TYPE MNG_RawDatagram :
STRUCT
	/// datagram header 
	Header: MNG_DatagramHeader;
	Payload: MNG_DataARRAY;
END_STRUCT
END_TYPE

(* stored: Version 1.1.0.1, ProductVersion 3.1.0.25
   DUT MNG_RawDatagram: Id {19952299-2866-4072-a49f-a6eac3909c1a} *)
